{attribute 'qualified_only}
PROGRAM COMM_FANUC

VAR_INPUT    
	arrf_Internal_FANUC_Input_1			: REAL;
	arrf_Internal_FANUC_Output_1		: UINT;
	
END_VAR

VAR_OUTPUT	
	
	sOutput_String						: STRING;
END_VAR

VAR		
	arrf_Internal_FANUC_TCP_xyz			: ARRAY [1..3] OF REAL;
	arrf_Internal_FANUC_TCP_uvw			: ARRAY [1..3] OF REAL;
	arrf_Internal_FANUC_TCP_Joints		: ARRAY [1..6] OF REAL;	
	fbCOMPARE_HEXA: COMPARE_HEXA;
END_VAR

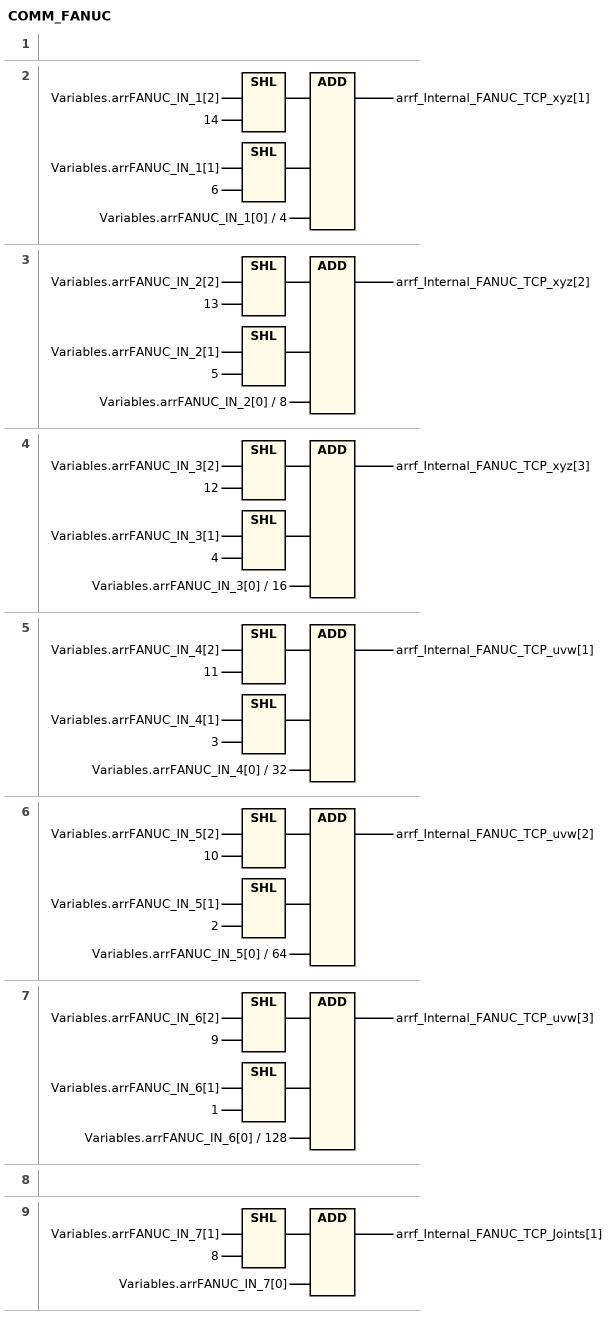
// NETWORK 1

// NETWORK 2
arrf_Internal_FANUC_TCP_xyz[1] := SHL(Variables.arrFANUC_IN_1[2], 14) + SHL(Variables.arrFANUC_IN_1[1], 6) + (Variables.arrFANUC_IN_1[0] / 4);

// NETWORK 3
arrf_Internal_FANUC_TCP_xyz[2] := SHL(Variables.arrFANUC_IN_2[2], 13) + SHL(Variables.arrFANUC_IN_2[1], 5) + (Variables.arrFANUC_IN_2[0] / 8);

// NETWORK 4
arrf_Internal_FANUC_TCP_xyz[3] := SHL(Variables.arrFANUC_IN_3[2], 12) + SHL(Variables.arrFANUC_IN_3[1], 4) + (Variables.arrFANUC_IN_3[0] / 16);

// NETWORK 5
arrf_Internal_FANUC_TCP_uvw[1] := SHL(Variables.arrFANUC_IN_4[2], 11) + SHL(Variables.arrFANUC_IN_4[1], 3) + (Variables.arrFANUC_IN_4[0] / 32);

// NETWORK 6
arrf_Internal_FANUC_TCP_uvw[2] := SHL(Variables.arrFANUC_IN_5[2], 10) + SHL(Variables.arrFANUC_IN_5[1], 2) + (Variables.arrFANUC_IN_5[0] / 64);

// NETWORK 7
arrf_Internal_FANUC_TCP_uvw[3] := SHL(Variables.arrFANUC_IN_6[2], 9) + SHL(Variables.arrFANUC_IN_6[1], 1) + (Variables.arrFANUC_IN_6[0] / 128);

// NETWORK 8

// NETWORK 9
arrf_Internal_FANUC_TCP_Joints[1] := SHL(Variables.arrFANUC_IN_7[1], 8) + Variables.arrFANUC_IN_7[0];

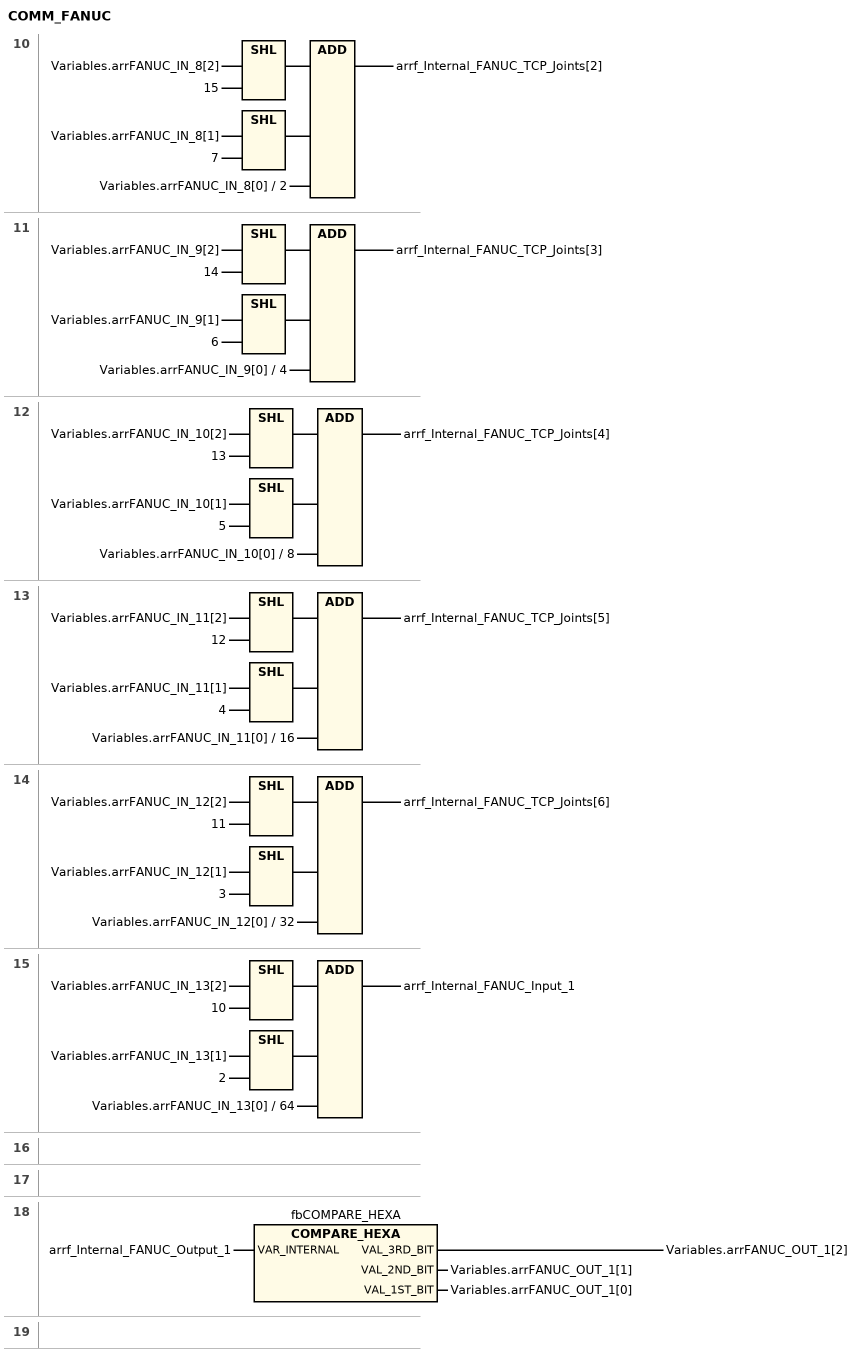
// NETWORK 10
arrf_Internal_FANUC_TCP_Joints[2] := SHL(Variables.arrFANUC_IN_8[2], 15) + SHL(Variables.arrFANUC_IN_8[1], 7) + (Variables.arrFANUC_IN_8[0] / 2);

// NETWORK 11
arrf_Internal_FANUC_TCP_Joints[3] := SHL(Variables.arrFANUC_IN_9[2], 14) + SHL(Variables.arrFANUC_IN_9[1], 6) + (Variables.arrFANUC_IN_9[0] / 4);

// NETWORK 12
arrf_Internal_FANUC_TCP_Joints[4] := SHL(Variables.arrFANUC_IN_10[2], 13) + SHL(Variables.arrFANUC_IN_10[1], 5) + (Variables.arrFANUC_IN_10[0] / 8);

// NETWORK 13
arrf_Internal_FANUC_TCP_Joints[5] := SHL(Variables.arrFANUC_IN_11[2], 12) + SHL(Variables.arrFANUC_IN_11[1], 4) + (Variables.arrFANUC_IN_11[0] / 16);

// NETWORK 14
arrf_Internal_FANUC_TCP_Joints[6] := SHL(Variables.arrFANUC_IN_12[2], 11) + SHL(Variables.arrFANUC_IN_12[1], 3) + (Variables.arrFANUC_IN_12[0] / 32);

// NETWORK 15
arrf_Internal_FANUC_Input_1 := SHL(Variables.arrFANUC_IN_13[2], 10) + SHL(Variables.arrFANUC_IN_13[1], 2) + (Variables.arrFANUC_IN_13[0] / 64);

// NETWORK 16

// NETWORK 17

// NETWORK 18
fbCOMPARE_HEXA(
    VAR_INTERNAL := arrf_Internal_FANUC_Output_1,
    VAL_2ND_BIT => Variables.arrFANUC_OUT_1[1],
    VAL_1ST_BIT => Variables.arrFANUC_OUT_1[0]); // COMPARE_HEXA
Variables.arrFANUC_OUT_1[2] := fbCOMPARE_HEXA.VAL_3RD_BIT;

// NETWORK 19

END_PROGRAM

(* stored: Version 1.1.0.1, ProductVersion 3.1.4024.0
   POU COMM_FANUC: Id {8a76c5d6-6bca-4661-83d7-85b058b2d811}, SpecialFunc None *)
